Staubli VAL3: HIT_YD.dtx

aio aConvSpeed = {link=ModbusSrv-0\Modbus-Word\ao[3]}
aio aPlcCmd = {link=ModbusSrv-0\Modbus-Word\ai[0]}
aio aRbAlarm = {link=ModbusSrv-0\Modbus-Word\ao[0]}
aio aRbStatus = {link=ModbusSrv-0\Modbus-Word\ao[1]}
bool _bConvExist = true
bool _bEndCycle
bool _bIsPicking = true
bool _bIsPlacing
bool _bMutexCnvQueue = true
bool _bOverflowed = true
bool _bPartInTool
bool _bSentToHome = true
bool _bVisionOK = true
bool bLockPage
bool bPickDetection
bool bSetConvSpeed
bool bSyn
bool bTransferData = true
dio dAlarm[8]
  [0] = {link=ModbusSrv-0\Modbus-Bit\do[8]}
  [1] = {link=ModbusSrv-0\Modbus-Bit\do[9]}
  [2] = {link=ModbusSrv-0\Modbus-Bit\do[10]}
  [3] = {link=ModbusSrv-0\Modbus-Bit\do[11]}
  [4] = {link=ModbusSrv-0\Modbus-Bit\do[12]}
  [5] = {link=ModbusSrv-0\Modbus-Bit\do[13]}
  [6] = {link=ModbusSrv-0\Modbus-Bit\do[14]}
  [7] = {link=ModbusSrv-0\Modbus-Bit\do[15]}
dio dBlow = {link=BasicIO-1\%Q5}
dio dConvControl[2]
  [0] = {link=BasicIO-1\%I4}
  [1] = {link=BasicIO-1\%Q6}
dio dPartInTool = {link=fIn0}
dio dPermitPlace[4]
  [0] = {link=BasicIO-1\%I3}
  [1] = {link=BasicIO-1\%I2}
  [2] = {link=BasicIO-1\%I1}
  [3] = {link=BasicIO-1\%I0}
dio dPlaceDone[4]
  [0] = {link=BasicIO-1\%Q11}
  [1] = {link=BasicIO-1\%Q10}
  [2] = {link=BasicIO-1\%Q9}
  [3] = {link=BasicIO-1\%Q8}
dio dStartControl[4]
  [0] = {link=ModbusSrv-0\Modbus-Bit\di[4]}
  [1] = {link=ModbusSrv-0\Modbus-Bit\di[5]}
  [2] = {link=ModbusSrv-0\Modbus-Bit\di[6]}
  [3] = {link=ModbusSrv-0\Modbus-Bit\di[7]}
dio dStartState[4]
  [0] = {link=ModbusSrv-0\Modbus-Bit\do[4]}
  [1] = {link=ModbusSrv-0\Modbus-Bit\do[5]}
  [2] = {link=ModbusSrv-0\Modbus-Bit\do[6]}
  [3] = {link=ModbusSrv-0\Modbus-Bit\do[7]}
dio dVacuum = {link=BasicIO-1\%Q4}
frame fConveyor = {x=365.904087, y=326.91934, z=-82.602337, rx=-0.010861, ry=-0.059106, rz=0.004608, fatherId=world[0]}
frame fDetection = {x=392.598601, y=461.346273, z=-82.976862, rx=0.205045, ry=0.617271, rz=0.011036, fatherId=world[0]}
jointRs jDropPart = {j1=102.785955, j2=-95.43121, j3=69.578977, j4=134.260732}
jointRs jHome = {j1=102.785955, j2=-95.43121, j3=69.578977, j4=134.260732}
jointRs jPark = {j1=102.785955, j2=-95.43121, j3=69.578977, j4=134.260732}
mdesc _mLoad = {accel=98.01, vel=99, decel=98.01, leave=40, reach=40}
mdesc mLoad = {accel=121, vel=110, decel=121, leave=40, reach=40}
mdesc mNomSpeed = {accel=121, vel=110, decel=121, leave=20, reach=20}
mdesc mPickDown = {accel=144, vel=120, decel=144, blend=off, leave=10, reach=10}
mdesc mPickup = {accel=121, vel=110, decel=121, leave=40, reach=40}
mdesc mPlaceDown = {accel=144, vel=120, decel=144, blend=off, leave=15, reach=15}
mdesc mPlaceUp = {accel=169, vel=130, decel=169, blend=cartesian, leave=30, reach=30}
mdesc mSlow = {accel=1, vel=10, decel=1, leave=10, reach=10}
mdesc mUnload = {accel=121, vel=110, decel=121, leave=40, reach=40}
num _nBlowDelay
num _nCntBypassed = 1
num _nCntPartsDone[2]
  [0] = 234927
  [1] = 234852
num _nCntTransfered = 2732
num _nConvSpd = 482.240758
num _nCycleTime[4]
  [0] = 2.619
  [1] = 0.715
  [2] = 2.425
  [3] = 0.561
num _nCycleTimeIndx = 2
num _nID = 1
num _nLastStateCMD
num _nOmacStat = 3
num _nPartID = 1
num _nPlaceCurItem[2]
num _nPullIndexTQ = 32
num _nPushIndexTQ = 32
num _nStateCMD
num _nTimer = 6773.495
num _nTrackErr = 334
num nBlowID = 0.4
num nBypass = 1
num nLoadRatio[4]
  [0] = 0.85
  [1] = 0.9
  [2] = 0.9
  [3] = 1
num nNomConvSpeed = 100
num nPartHeight = 5
num nPickAppro = 65
num nPickOS_X
num nPickOS_Y = 2
num nPlaceAppro = 60
public num nPlaceNum
num nSafeMaxX = 850
num nSafeMaxY = 650
num nSafeMinX
num nSafeMinY
num nStopTime
num nTestData[5]
  [0] = 6
  [1] = -49
  [2] = 55
  [4] = 184151
num nVacuumID = 0.1
num nWaitDist2Up4BP = -300
num nWaitDistToDown = 50
num nWaitDistToUp[1 3]
  [0,0] = -80
  [0,1] = 120
  [0,2] = 400
num nWaitDistX
object _oTransferQueue[1 100]
  [0,0]
    num nID = -1
    num nLatchedValue
    trsf trTrsf
  [0,1]
    num nID = -1
    num nLatchedValue
    trsf trTrsf
  [0,2]
    num nID = -1
    num nLatchedValue
    trsf trTrsf
  [0,3]
    num nID = -1
    num nLatchedValue
    trsf trTrsf
  [0,4]
    num nID = -1
    num nLatchedValue
    trsf trTrsf
  [0,5]
    num nID = -1
    num nLatchedValue
    trsf trTrsf
  [0,6]
    num nID = -1
    num nLatchedValue
    trsf trTrsf
  [0,7]
    num nID = -1
    num nLatchedValue
    trsf trTrsf
  [0,8]
    num nID = -1
    num nLatchedValue
    trsf trTrsf
  [0,9]
    num nID = -1
    num nLatchedValue
    trsf trTrsf
  [0,10]
    num nID = -1
    num nLatchedValue
    trsf trTrsf
  [0,11]
    num nID = -1
    num nLatchedValue
    trsf trTrsf
  [0,12]
    num nID = -1
    num nLatchedValue
    trsf trTrsf
  [0,13]
    num nID = -1
    num nLatchedValue
    trsf trTrsf
  [0,14]
    num nID = -1
    num nLatchedValue
    trsf trTrsf
  [0,15]
    num nID = -1
    num nLatchedValue
    trsf trTrsf
  [0,16]
    num nID = -1
    num nLatchedValue
    trsf trTrsf
  [0,17]
    num nID = -1
    num nLatchedValue
    trsf trTrsf
  [0,18]
    num nID = -1
    num nLatchedValue
    trsf trTrsf
  [0,19]
    num nID = -1
    num nLatchedValue
    trsf trTrsf
  [0,20]
    num nID = -1
    num nLatchedValue
    trsf trTrsf
  [0,21]
    num nID = -1
    num nLatchedValue
    trsf trTrsf
  [0,22]
    num nID = -1
    num nLatchedValue
    trsf trTrsf
  [0,23]
    num nID = -1
    num nLatchedValue
    trsf trTrsf
  [0,24]
    num nID = -1
    num nLatchedValue
    trsf trTrsf
  [0,25]
    num nID = -1
    num nLatchedValue
    trsf trTrsf
  [0,26]
    num nID = -1
    num nLatchedValue
    trsf trTrsf
  [0,27]
    num nID = -1
    num nLatchedValue
    trsf trTrsf
  [0,28]
    num nID = -1
    num nLatchedValue
    trsf trTrsf
  [0,29]
    num nID = -1
    num nLatchedValue
    trsf trTrsf
  [0,30]
    num nID = -1
    num nLatchedValue
    trsf trTrsf
  [0,31]
    num nID = -1
    num nLatchedValue
    trsf trTrsf
  [0,32]
    num nID = -1
    num nLatchedValue
    trsf trTrsf
  [0,33]
    num nID = -1
    num nLatchedValue
    trsf trTrsf
  [0,34]
    num nID = -1
    num nLatchedValue
    trsf trTrsf
  [0,35]
    num nID = -1
    num nLatchedValue
    trsf trTrsf
  [0,36]
    num nID = -1
    num nLatchedValue
    trsf trTrsf
  [0,37]
    num nID = -1
    num nLatchedValue
    trsf trTrsf
  [0,38]
    num nID = -1
    num nLatchedValue
    trsf trTrsf
  [0,39]
    num nID = -1
    num nLatchedValue
    trsf trTrsf
  [0,40]
    num nID = -1
    num nLatchedValue
    trsf trTrsf
  [0,41]
    num nID = -1
    num nLatchedValue
    trsf trTrsf
  [0,42]
    num nID = -1
    num nLatchedValue
    trsf trTrsf
  [0,43]
    num nID = -1
    num nLatchedValue
    trsf trTrsf
  [0,44]
    num nID = -1
    num nLatchedValue
    trsf trTrsf
  [0,45]
    num nID = -1
    num nLatchedValue
    trsf trTrsf
  [0,46]
    num nID = -1
    num nLatchedValue
    trsf trTrsf
  [0,47]
    num nID = -1
    num nLatchedValue
    trsf trTrsf
  [0,48]
    num nID = -1
    num nLatchedValue
    trsf trTrsf
  [0,49]
    num nID = -1
    num nLatchedValue
    trsf trTrsf
  [0,50]
    num nID = -1
    num nLatchedValue
    trsf trTrsf
  [0,51]
    num nID = -1
    num nLatchedValue
    trsf trTrsf
  [0,52]
    num nID = -1
    num nLatchedValue
    trsf trTrsf
  [0,53]
    num nID = -1
    num nLatchedValue
    trsf trTrsf
  [0,54]
    num nID = -1
    num nLatchedValue
    trsf trTrsf
  [0,55]
    num nID = -1
    num nLatchedValue
    trsf trTrsf
  [0,56]
    num nID = -1
    num nLatchedValue
    trsf trTrsf
  [0,57]
    num nID = -1
    num nLatchedValue
    trsf trTrsf
  [0,58]
    num nID = -1
    num nLatchedValue
    trsf trTrsf
  [0,59]
    num nID = -1
    num nLatchedValue
    trsf trTrsf
  [0,60]
    num nID = -1
    num nLatchedValue
    trsf trTrsf
  [0,61]
    num nID = -1
    num nLatchedValue
    trsf trTrsf
  [0,62]
    num nID = -1
    num nLatchedValue
    trsf trTrsf
  [0,63]
    num nID = -1
    num nLatchedValue
    trsf trTrsf
  [0,64]
    num nID = -1
    num nLatchedValue
    trsf trTrsf
  [0,65]
    num nID = -1
    num nLatchedValue
    trsf trTrsf
  [0,66]
    num nID = -1
    num nLatchedValue
    trsf trTrsf
  [0,67]
    num nID = -1
    num nLatchedValue
    trsf trTrsf
  [0,68]
    num nID = -1
    num nLatchedValue
    trsf trTrsf
  [0,69]
    num nID = -1
    num nLatchedValue
    trsf trTrsf
  [0,70]
    num nID = -1
    num nLatchedValue
    trsf trTrsf
  [0,71]
    num nID = -1
    num nLatchedValue
    trsf trTrsf
  [0,72]
    num nID = -1
    num nLatchedValue
    trsf trTrsf
  [0,73]
    num nID = -1
    num nLatchedValue
    trsf trTrsf
  [0,74]
    num nID = -1
    num nLatchedValue
    trsf trTrsf
  [0,75]
    num nID = -1
    num nLatchedValue
    trsf trTrsf
  [0,76]
    num nID = -1
    num nLatchedValue
    trsf trTrsf
  [0,77]
    num nID = -1
    num nLatchedValue
    trsf trTrsf
  [0,78]
    num nID = -1
    num nLatchedValue
    trsf trTrsf
  [0,79]
    num nID = -1
    num nLatchedValue
    trsf trTrsf
  [0,80]
    num nID = -1
    num nLatchedValue
    trsf trTrsf
  [0,81]
    num nID = -1
    num nLatchedValue
    trsf trTrsf
  [0,82]
    num nID = -1
    num nLatchedValue
    trsf trTrsf
  [0,83]
    num nID = -1
    num nLatchedValue
    trsf trTrsf
  [0,84]
    num nID = -1
    num nLatchedValue
    trsf trTrsf
  [0,85]
    num nID = -1
    num nLatchedValue
    trsf trTrsf
  [0,86]
    num nID = -1
    num nLatchedValue
    trsf trTrsf
  [0,87]
    num nID = -1
    num nLatchedValue
    trsf trTrsf
  [0,88]
    num nID = -1
    num nLatchedValue
    trsf trTrsf
  [0,89]
    num nID = -1
    num nLatchedValue
    trsf trTrsf
  [0,90]
    num nID = -1
    num nLatchedValue
    trsf trTrsf
  [0,91]
    num nID = -1
    num nLatchedValue
    trsf trTrsf
  [0,92]
    num nID = -1
    num nLatchedValue
    trsf trTrsf
  [0,93]
    num nID = -1
    num nLatchedValue
    trsf trTrsf
  [0,94]
    num nID = -1
    num nLatchedValue
    trsf trTrsf
  [0,95]
    num nID = -1
    num nLatchedValue
    trsf trTrsf
  [0,96]
    num nID = -1
    num nLatchedValue
    trsf trTrsf
  [0,97]
    num nID = -1
    num nLatchedValue
    trsf trTrsf
  [0,98]
    num nID = -1
    num nLatchedValue
    trsf trTrsf
  [0,99]
    num nID = -1
    num nLatchedValue
    trsf trTrsf
pointRs pPick = {x=51.000306, y=-30.000014, z=4.992462, rx=0, ry=0, rz=112.9, shoulder=lefty, fatherId=fDetection[0]}
pointRs pPlace[4]
  [0] = {x=360, y=110, z=-83, rx=180, ry=0, rz=-100, shoulder=lefty, fatherId=world[0]}
  [1] = {x=490, y=105, z=-83, rx=180, ry=0, rz=-100, shoulder=lefty, fatherId=world[0]}
  [2] = {x=620, y=105, z=-83, rx=180, rz=-98.02183, shoulder=lefty, fatherId=world[0]}
  [3] = {x=760, y=105, z=-83, rx=180, rz=-98.02084, shoulder=lefty, fatherId=world[0]}
sio skToRobot = {link=Socket\toRobot_sk1}
sio sktoPC = {link=Socket\toPC}
sio synServer = {link=Socket\synRobot1}
string _sCycleStatus = "Distance to pick: -359.23"
string sConveyorList = "cvIn"
string sDataPC = "run"
string sString = "done"
tool tGripper = {z=85, rz=45, fatherId=flange[0], ioLink=valve1}
